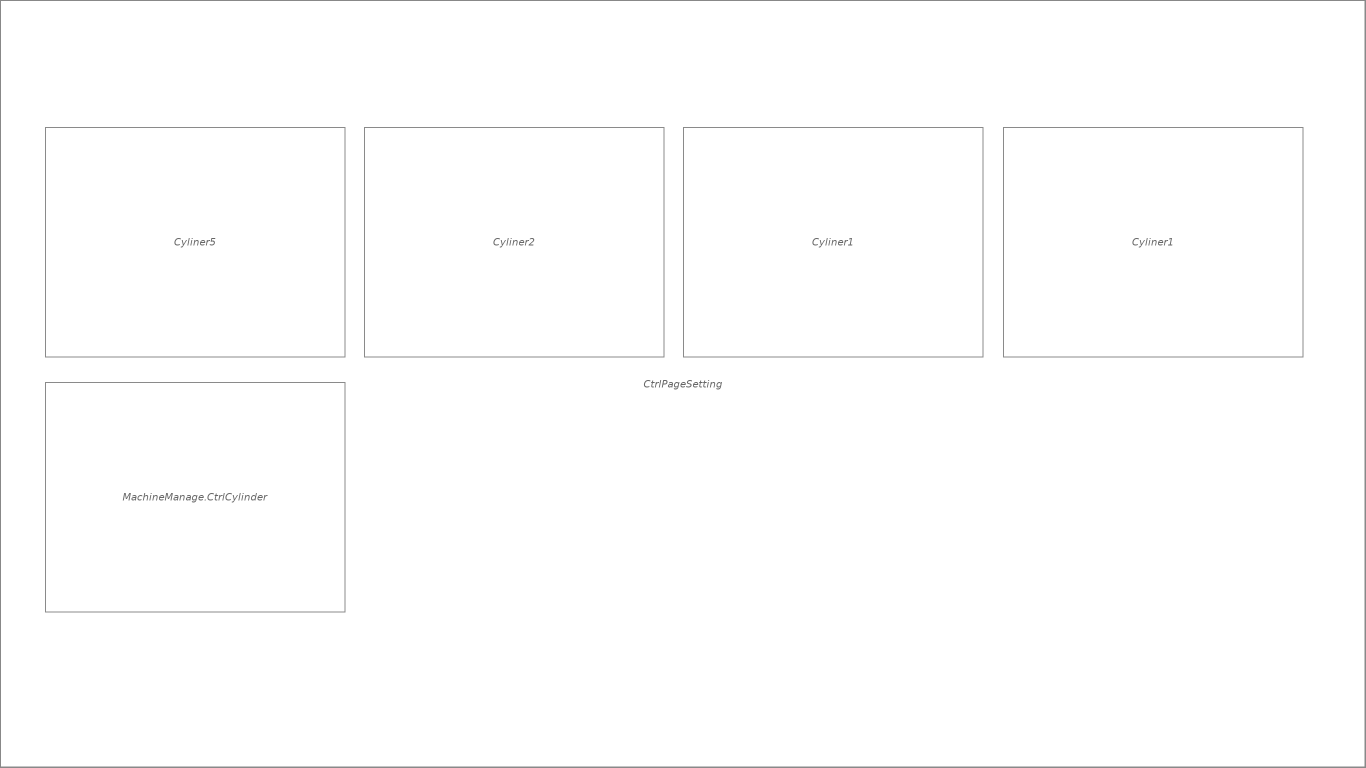
VISUALIZATION PageSetting_TakeUc_M  // 1366x768
    Frame (0,0 1366x768)
        shows CtrlPageSetting()
    Frame (364,127 300x230)
        shows Cyliner2(System := G_stSystem, Cylinder := G_arrCylinder[E_Cylinder.TakeUc1Y], CylinderData := G_arrCylinderData[E_Cylinder.TakeUc1Y])
    Frame (683,127 300x230)
        shows Cyliner1(System := G_stSystem, Cylinder := G_arrCylinder[E_Cylinder.TakeUc1Z1], CylinderData := G_arrCylinderData[E_Cylinder.TakeUc1Z1])
    Frame (1003,127 300x230)
        shows Cyliner1(System := G_stSystem, Cylinder := G_arrCylinder[E_Cylinder.TakeUc1Z2], CylinderData := G_arrCylinderData[E_Cylinder.TakeUc1Z2])
    Frame (45,382 300x230)
        shows MachineManage.CtrlCylinder(System := G_stSystem, Cylinder := G_arrCylinder[E_Cylinder.TakeUc1Rotate], CylinderData := G_arrCylinderData[E_Cylinder.TakeUc1Rotate])
    Frame (45,127 300x230)
        shows Cyliner5(System := G_stSystem, Cylinder := G_arrCylinder[E_Cylinder.TakeUc1Clamp], CylinderData := G_arrCylinderData[E_Cylinder.TakeUc1Clamp])
END_VISUALIZATION

(* stored: Version 1.1.0.1, ProductVersion 3.1.4024.3
   Visu PageSetting_TakeUc_M: Id {42d4b046-9f01-4ddc-9c22-e783fc7b57c9} *)
